FUNCTION_BLOCK VltProbe_Mem
VAR
	a : BOOL;
	b : BOOL;
	out : BOOL;
END_VAR

out := a;

ACTION A_G:
out := a AND b;
END_ACTION

PROPERTY P_G : BOOL
GET
P_G := a AND b;
END_GET
SET
out := P_G;
END_SET
END_PROPERTY

END_FUNCTION_BLOCK
